// TIA Portal V19 export
DATA_BLOCK "Sample_alarmed_FB_DB_1"   // DB2
// stored: InstanceOfName Sample_alarmed_FB, InstanceOfType FB
"Sample_alarmed_FB"
   // VAR_INPUT
   //    Alarm_Trigger : Bool;
   //    Timer_PT : Time;
   //    ACK_Button : Bool;
   //    Reset_Button : Bool;
   // END_VAR
   // VAR_OUTPUT
   //    Alarm : Bool;
   //    Alarm_ACKED : Bool;
   //    Alarm_Indicator : Bool;
   // END_VAR
   // VAR
   //    Alarm_Timer { S7_SetPoint := 'True'} : TON_TIME;
   //    Alarm_Timer_Done : Bool;
   //    Alarm_Active : Bool;
   //    Alarm_ACK : Bool;
   //    Alarm_Reset : Bool;
   // END_VAR
BEGIN
END_DATA_BLOCK
